// TIA Portal V17 export
// export: Created 2026-04-13T11:12:03.850624Z, ExportSetting WithDefaults, DisplayName Totally Integrated Automation Portal, DisplayVersion V17 Update 4, DisplayName TIA Portal Openness, DisplayVersion V17 Update 4, DisplayName TIA Portal Version Control Interface, DisplayVersion V17, DisplayName SINAMICS Startdrive Advanced, DisplayVersion V17, DisplayName SINAMICS Startdrive G130, G150, S120, S150, SINAMICS MV, S210, DisplayVersion V17, DisplayName SINAMICS Startdrive G110M, G120, G120C, G120D, G120P, G115D, DisplayVersion V17, DisplayName STEP 7 Professional, DisplayVersion V17 Update 4, DisplayName STEP 7 Safety, DisplayVersion V17, DisplayName WinCC Professional, DisplayVersion V17 Update 4
FUNCTION_BLOCK "A1-阀带反馈"   // FB18, SCL
{ S7_Optimized_Access := 'TRUE' }
VERSION : 0.1
// stored: AutoNumber true, IsIECCheckEnabled false, IsRetainMemResEnabled false, MemoryReserve 100, SetENOAutomatically false, UDAEnableTagReadback false
   VAR
      泄压阀 { S7_SetPoint := 'True'} : "A3-普通阀控制";
      进风冷却水阀 { S7_SetPoint := 'True'} : "A3-普通阀控制";
      输送进风阀 { S7_SetPoint := 'True'} : "A3-普通阀控制";
      气流雾化阀 { S7_SetPoint := 'True'} : "A3-普通阀控制";
      开式排风隔断阀 { S7_SetPoint := 'True'} : "A3-普通阀控制";
      闭式排风隔断阀 { S7_SetPoint := 'True'} : "A3-普通阀控制";
      开式进风隔断阀 { S7_SetPoint := 'True'} : "A3-普通阀控制";
      闭式进风隔断阀 { S7_SetPoint := 'True'} : "A3-普通阀控制";
      一级冷却水阀 { S7_SetPoint := 'True'} : "A3-普通阀控制";
      二级冷冻水阀 { S7_SetPoint := 'True'} : "A3-普通阀控制";
      一级排液阀 { S7_SetPoint := 'True'} : "A3-普通阀控制";
      二级排液阀 { S7_SetPoint := 'True'} : "A3-普通阀控制";
      除雾排液阀 { S7_SetPoint := 'True'} : "A3-普通阀控制";
      补氮阀 : "A3-普通阀控制";
      进氮阀 { S7_SetPoint := 'True'} : "A3-普通阀控制";
      塔顶清洗球阀 { S7_SetPoint := 'True'} : "A3-普通阀控制";
      溶剂回收排放阀 { S7_SetPoint := 'True'} : "A3-普通阀控制";
      室内排水隔膜泵 { S7_SetPoint := 'True'} : "A3-普通阀控制";
      溶剂排液泵 { S7_SetPoint := 'True'} : "A3-普通阀控制";
      清洗伸缩气缸 { S7_SetPoint := 'True'} : "A3-普通阀控制";
   END_VAR
BEGIN
   REGION 带反馈控制阀
      // "ALQ冷却水流量低报警"



       IF "MJF进风加热比例调节阀" THEN
           "QJF进风蒸汽比例调节阀" := 1;
       ELSE
           "QJF进风蒸汽比例调节阀" := 0;
       END_IF;

       IF "MJF进风蒸汽开关阀" THEN
           "QJF进风蒸汽开关阀" := 1;
       ELSE
           "QJF进风蒸汽开关阀" := 0;
       END_IF;

       IF "MJF进风蒸汽排水阀" THEN
           "QJF进风蒸汽排水阀" := 1;
       ELSE
           "QJF进风蒸汽排水阀" := 0;
       END_IF;

       IF "MHF回风蒸汽排水阀" THEN
           "QHF回风蒸汽排水阀" := 1;
       ELSE
           "QHF回风蒸汽排水阀" :=0;
       END_IF;



           IF "MSF输送风机" THEN
               "QSS输送风机" := 1;
           ELSE
               "QSS输送风机" := 0;
           END_IF;


           IF "MRJ溶剂排液泵" THEN
               "QRJ溶剂排液泵" := 1;
           ELSE
               "QRJ溶剂排液泵" := 0;
           END_IF;


           IF "MSN室内排水隔膜泵" THEN
               "QSN室内排水隔膜泵" := 1;
           ELSE
               "QSN室内排水隔膜泵" := 0;
           END_IF;


           IF "MCC除尘脉冲" THEN
               "QCC除尘脉冲" := 1;
           ELSE
               "QCC除尘脉冲" := 0;
           END_IF;



           #泄压阀(模式设定 := "PW".MS模式设定,
                条件1 := 0.0,
                条件2 := 0.0,
                阀开信号 := "IXY泄压阀开反馈",
                阀关信号 := "IXY泄压阀关反馈",
                手动控制按钮开 := "MXY泄压阀",
                阀状态 := "QXY泄压阀",
                阀开报警 := "AXY泄压阀开报警",
                阀关报警 := "AXY泄压阀关报警");

           #进风冷却水阀(模式设定 := "PW".MS模式设定,
                   条件1 := 0.0,
                   条件2 := 0.0,
                   阀开信号 := "IJF进风冷却水阀开反馈",
                   阀关信号 := "IJF进风冷却水阀关反馈",
                   手动控制按钮开 := "MJF进风冷却水阀",
                   阀状态 := "QJF进风冷却水阀",
                   阀开报警 := "AJF进风冷却水阀开报警",
                   阀关报警 := "AJF进风冷却水阀关报警");

           #输送进风阀(模式设定 := "PW".MS模式设定,
                  条件1 := 0.0,
                  条件2 := 0.0,
                  阀开信号 := "ISF输送进风阀开反馈",
                  阀关信号 := "ISF输送进风阀关反馈",
                  手动控制按钮开 := "MSS输送进风阀",
                  阀状态 := "QSS输送进风阀",
                  阀开报警 := "ASS输送进风阀开报警",
                  阀关报警 := "ASS输送进风阀关报警");

           #气流雾化阀(模式设定 := "PW".MS模式设定,
                  条件1 := 0.0,
                  条件2 := 0.0,
                  阀开信号 := "IQL气流雾化阀开反馈",
                  阀关信号 := "IQL气流雾化阀关反馈",
                  手动控制按钮开 := "MQL气流雾化阀",
                  阀状态 := "QQL气流雾化阀",
                  阀开报警 := "AQL气流雾化阀开报警",
                  阀关报警 := "AQL气流雾化阀关报警");


           #开式排风隔断阀(模式设定 := "PW".MS模式设定,
                    条件1 := 0.0,
                    条件2 := 0.0,
                    阀开信号 := "IKS开式排风隔断阀开反馈",
                    阀关信号 := "IKS开式排风隔断阀关反馈",
                    手动控制按钮开 := "MKS开式排风隔断阀",
                    阀状态 := "QKS开式排风隔断阀",
                    阀开报警 := "AKS开式排风隔断阀开报警",
                    阀关报警 := "AKS开式排风隔断阀关报警");

           #闭式排风隔断阀(模式设定 := "PW".MS模式设定,
                    条件1 := 0.0,
                    条件2 := 0.0,
                    阀开信号 := "IBS闭式排风隔断阀开反馈",
                    阀关信号 := "IBS闭式排风隔断阀关反馈",
                    手动控制按钮开 := "MBS闭式排风隔断阀",
                    阀状态 := "QBS闭式排风隔断阀",
                    阀开报警 := "ABS闭式排风隔断阀开报警",
                    阀关报警 := "ABS闭式排风隔断阀关报警");

           #开式进风隔断阀(模式设定 := "PW".MS模式设定,
                    条件1 := 0.0,
                    条件2 := 0.0,
                    阀开信号 := "IKS开式进风隔断阀开反馈",
                    阀关信号 := "IKS开式进风隔断阀关反馈",
                    手动控制按钮开 := "MKS开式进风隔断阀",
                    阀状态 := "QKS开式进风隔断阀",
                    阀开报警 := "AKS开式进风隔断阀开报警",
                    阀关报警 := "AKS开式进风隔断阀关报警");


           #闭式进风隔断阀(模式设定 := "PW".MS模式设定,
                    条件1 := 0.0,
                    条件2 := 0.0,
                    阀开信号 := "IBS闭式进风隔断阀开反馈",
                    阀关信号 := "IBS闭式进风隔断阀关反馈",
                    手动控制按钮开 := "MBS闭式进风隔断阀",
                    阀状态 := "QBS闭式进风隔断阀",
                    阀开报警 := "ABS闭式进风隔断阀开报警",
                    阀关报警 := "ABS闭式进风隔断阀关报警");

           #一级冷却水阀(模式设定 := "PW".MS模式设定,
                   条件1 := 0.0,
                   条件2 := 0.0,
                   阀开信号 := "IYJ一级冷却水阀开反馈",
                   阀关信号 := "IYJ一级冷却水阀关反馈",
                   手动控制按钮开 := "MYJ一级冷却水阀",
                   阀状态 := "QYJ一级冷却水阀",
                   阀开报警 := "AYJ一级冷却水阀开报警",
                   阀关报警 := "AYJ一级冷却水阀关报警");


           #二级冷冻水阀(模式设定 := "PW".MS模式设定,//Q点不对
                   条件1 := 0.0,
                   条件2 := 0.0,
                   阀开信号 := "IEJ二级冷冻水阀开反馈",
                   阀关信号 := "IEJ二级冷冻水阀关反馈",
                   手动控制按钮开 := "MEJ二级冷冻水阀",
                   阀状态 := "QEJ二级冷冻水阀",
                   阀开报警 := "AEJ二级冷冻水阀开报警",
                   阀关报警 := "AEJ二级冷冻水阀关报警");

           #一级排液阀(模式设定 := "PW".MS模式设定,
                  条件1 := 0.0,
                  条件2 := 0.0,
                  阀开信号 := "IYJ一级排液阀开反馈",
                  阀关信号 := "IYJ一级排液阀关反馈",
                  手动控制按钮开 := "MYJ一级排液阀",
                  阀状态 := "QYJ一级排液阀",
                  阀开报警 := "AYJ一级排液阀开报警",
                  阀关报警 := "AYJ一级排液阀关报警");


           #二级排液阀(模式设定 := "PW".MS模式设定,
                  条件1 := 0.0,
                  条件2 := 0.0,
                  阀开信号 := "IEJ二级排液阀开反馈",
                  阀关信号 := "IEJ二级排液阀关反馈",
                  手动控制按钮开 := "MEJ二级排液阀",
                  阀状态 := "QEJ二级排液阀",
                  阀开报警 := "AEJ二级排液阀开报警",
                  阀关报警 := "AEJ二级排液阀关报警");

           #除雾排液阀(模式设定 := "PW".MS模式设定,
                  条件1 := 0.0,
                  条件2 := 0.0,
                  阀开信号 := "ICW除雾排液阀开反馈",
                  阀关信号 := "ICW除雾排液阀关反馈",
                  手动控制按钮开 := "MCW除雾排液阀",
                  阀状态 := "QCW除雾排液阀",
                  阀开报警 := "ACW除雾排液阀开报警",
                  阀关报警 := "ACW除雾排液阀关报警");

           #补氮阀(模式设定 := "PW".MS模式设定,
                条件1 := 0.0,
                条件2 := 0.0,
                阀开信号 := "IBD补氮阀开反馈",
                阀关信号 := "IBD补氮阀关反馈",
                手动控制按钮开 := "MBD补氮阀",
                阀状态 := "QBD补氮阀",
                阀开报警 := "ABD补氮阀开报警",
                阀关报警 := "ABD补氮阀关报警");

           #进氮阀(模式设定 := "PW".MS模式设定,
                条件1 := 0.0,
                条件2 := 0.0,
                阀开信号 := "IJD进氮阀开反馈",
                阀关信号 := "IJD进氮阀关反馈",
                手动控制按钮开 := "MJD进氮阀",
                阀状态 := "QJD进氮阀",
                阀开报警 := "AJD进氮阀开报警",
                阀关报警 := "AJD进氮阀关报警");


           #塔顶清洗球阀(模式设定 := "PW".MS模式设定,
                   条件1 := 0.0,
                   条件2 := 0.0,
                   阀开信号 := "ITD塔顶清洗球阀开反馈",
                   阀关信号 := "ITD塔顶清洗球阀关反馈",
                   手动控制按钮开 := "MTD塔顶清洗球阀",
                   阀状态 := "QTD塔顶清洗球阀",
                   阀开报警 := "ATD塔顶清洗球阀开报警",
                   阀关报警 := "ATD塔顶清洗球阀关报警");

           #溶剂回收排放阀(模式设定 := "PW".MS模式设定,
                    条件1 := 0.0,
                    条件2 := 0.0,
                    阀开信号 := "IRJ溶剂回收排放阀开反馈",
                    阀关信号 := "IRJ溶剂回收排放阀关反馈",
                    手动控制按钮开 := "MRJ溶剂回收排放阀",
                    阀状态 := "QRJ溶剂回收排放阀",
                    阀开报警 := "ARJ溶剂回收排放阀开报警",
                    阀关报警 := "ARJ溶剂回收排放阀关报警");


           #室内排水隔膜泵(模式设定 := "PW".MS模式设定,
                    条件1 := 0.0,
                    条件2 := 0.0,
                    阀开信号 := "ISN室内排水开反馈",
                    阀关信号 := "ISN室内排水关反馈",
                    手动控制按钮开 := "MSN室内排水隔膜泵",
                    阀状态 := "QSN室内排水隔膜泵",
                    阀开报警 := "ASN室内排水开反馈报警",
                    阀关报警 := "ASN室内排水关反馈报警");


           #溶剂排液泵(模式设定 := "PW".MS模式设定,
                  条件1 := 0.0,
                  条件2 := 0.0,
                  阀开信号 := "IRJ溶剂排液泵开反馈",
                  阀关信号 := "IRJ溶剂排液泵关反馈",
                  手动控制按钮开 := "MRJ溶剂排液泵",
                  阀状态 := "QRJ溶剂排液泵",
                  阀开报警 :="ARJ溶剂排液泵开报警" ,
                  阀关报警 := "ARJ溶剂排液泵关报警");



         (*  #清洗伸缩气缸(模式设定 := "PW".MS模式设定,
                  条件1 := 0.0,
                  条件2 := 0.0,
                  阀开信号 := "IQX清洗伸缩气缸开反馈",
                  阀关信号 := "IQX清洗伸缩气缸关反馈",

                  阀状态 := "QQG气缸升降阀",
                  阀开报警 := "AQX清洗伸缩气缸开报警",
                  阀关报警 := "AQX清洗伸缩气缸关报警"); *)


   END_REGION
END_FUNCTION_BLOCK
